TYPE sMC_CAM_REF :
STRUCT
	Distance:REAL;
	Phase:REAL;
END_STRUCT
END_TYPE

(* stored: Version 1.1.0.1, ProductVersion 3.1.4024.9
   DUT sMC_CAM_REF: Id {cfa860cb-7655-466f-a0cc-c0c8a35902ba} *)
